(* IEC 61131-3 sources: CodesysTest/alpha/export/FBs/Components/Aux IO/FB_OutputPulseManager.pou, 5 files *)

(* ---- FB_OutputPulseManager.pou.st ---- *)
(*#-#-#-#-#-#-#-#-#-#---Declaration---#-#-#-#-#-#-#-#-#-#-#-#-#*)

FUNCTION_BLOCK FINAL FB_OutputPulseManager
VAR_INPUT
END_VAR
VAR_OUTPUT
	configOut1 : BOOL;
	configOut2 : BOOL;
	configOut3 : BOOL;
	configOut4 : BOOL;
END_VAR
VAR
	_reset : BOOL;
	_configOutput1Pulse : FB_MonostableMultivibrator();
	_configOutput2Pulse : FB_MonostableMultivibrator();
	_configOutput3Pulse : FB_MonostableMultivibrator();
	_configOutput4Pulse : FB_MonostableMultivibrator();
END_VAR
(*#-#-#-#-#-#-#-#-#-#---Implementation---#-#-#-#-#-#-#-#-#-#-#-#-#*)

IF _reset THEN
	_reset := FALSE;
	_configOutput1Pulse.Reset();
	_configOutput2Pulse.Reset();
	_configOutput3Pulse.Reset();
	_configOutput4Pulse.Reset();
	_configOutput1Pulse.ManualOff();
	_configOutput2Pulse.ManualOff();
	_configOutput3Pulse.ManualOff();
	_configOutput4Pulse.ManualOff();
END_IF

// Pulse outputs that are temporary statuses (Cycle Complete) vs. held (Waiting for Printer)
_configOutput1Pulse(Q => configOut1);
_configOutput2Pulse(Q => configOut2);
_configOutput3Pulse(Q => configOut3);
_configOutput4Pulse(Q => configOut4);
_configOutput1Pulse.DwellSetting := 500;
_configOutput2Pulse.DwellSetting := 500;
_configOutput3Pulse.DwellSetting := 500;
_configOutput4Pulse.DwellSetting := 500;

(* ---- ManualOff.m.st ---- *)
(*#-#-#-#-#-#-#-#-#-#---Declaration---#-#-#-#-#-#-#-#-#-#-#-#-#*)

METHOD ManualOff
VAR_INPUT
	output : INT;
END_VAR
(*#-#-#-#-#-#-#-#-#-#---Implementation---#-#-#-#-#-#-#-#-#-#-#-#-#*)

CASE output OF
	1: _configOutput1Pulse.ManualOn();
	2: _configOutput2Pulse.ManualOn();
	3: _configOutput3Pulse.ManualOn();
	4: _configOutput4Pulse.ManualOn();
END_CASE

(* ---- ManualOn.m.st ---- *)
(*#-#-#-#-#-#-#-#-#-#---Declaration---#-#-#-#-#-#-#-#-#-#-#-#-#*)

METHOD ManualOn
VAR_INPUT
	output : INT;
END_VAR
(*#-#-#-#-#-#-#-#-#-#---Implementation---#-#-#-#-#-#-#-#-#-#-#-#-#*)

CASE output OF
	1: _configOutput1Pulse.ManualOff();
	2: _configOutput2Pulse.ManualOff();
	3: _configOutput3Pulse.ManualOff();
	4: _configOutput4Pulse.ManualOff();
END_CASE

(* ---- Reset.m.st ---- *)
(*#-#-#-#-#-#-#-#-#-#---Declaration---#-#-#-#-#-#-#-#-#-#-#-#-#*)

METHOD Reset
VAR_INPUT
END_VAR
(*#-#-#-#-#-#-#-#-#-#---Implementation---#-#-#-#-#-#-#-#-#-#-#-#-#*)

_reset := TRUE;

(* ---- Trigger.m.st ---- *)
(*#-#-#-#-#-#-#-#-#-#---Declaration---#-#-#-#-#-#-#-#-#-#-#-#-#*)

METHOD Trigger
VAR_INPUT
	output : INT;
END_VAR
(*#-#-#-#-#-#-#-#-#-#---Implementation---#-#-#-#-#-#-#-#-#-#-#-#-#*)

CASE output OF
	1: _configOutput1Pulse.Trigger();
	2: _configOutput2Pulse.Trigger();
	3: _configOutput3Pulse.Trigger();
	4: _configOutput4Pulse.Trigger();
END_CASE
